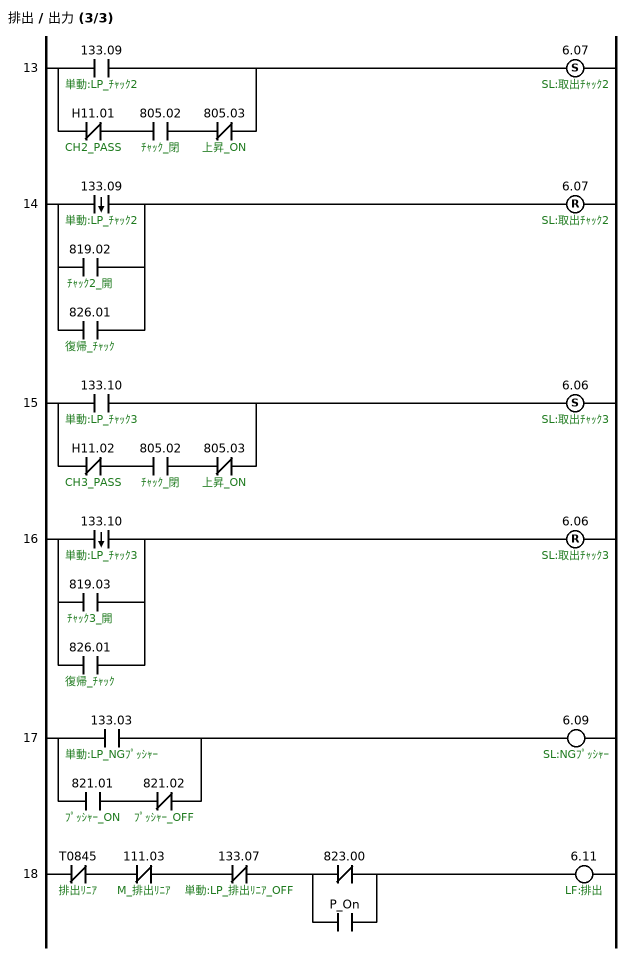
; [picture p192: 排出 / 出力, rungs 13-18]
; rung 13
LD 133.09  ; 単動:LP_ﾁｬｯｸ2
LDNOT H11.01  ; CH2_PASS
AND 805.02  ; ﾁｬｯｸ_閉
ANDNOT 805.03  ; 上昇_ON
ORLD
SET 6.07  ; SL:取出ﾁｬｯｸ2
; rung 14
%LD 133.09  ; 単動:LP_ﾁｬｯｸ2
OR 819.02  ; ﾁｬｯｸ2_開
OR 826.01  ; 復帰_ﾁｬｯｸ
RSET 6.07  ; SL:取出ﾁｬｯｸ2
; rung 15
LD 133.10  ; 単動:LP_ﾁｬｯｸ3
LDNOT H11.02  ; CH3_PASS
AND 805.02  ; ﾁｬｯｸ_閉
ANDNOT 805.03  ; 上昇_ON
ORLD
SET 6.06  ; SL:取出ﾁｬｯｸ3
; rung 16
%LD 133.10  ; 単動:LP_ﾁｬｯｸ3
OR 819.03  ; ﾁｬｯｸ3_開
OR 826.01  ; 復帰_ﾁｬｯｸ
RSET 6.06  ; SL:取出ﾁｬｯｸ3
; rung 17
LD 133.03  ; 単動:LP_NGﾌﾟｯｼｬｰ
LD 821.01  ; ﾌﾟｯｼｬｰ_ON
ANDNOT 821.02  ; ﾌﾟｯｼｬｰ_OFF
ORLD
OUT 6.09  ; SL:NGﾌﾟｯｼｬｰ
; rung 18
LDNOT T0845  ; 排出ﾘﾆｱ
ANDNOT 111.03  ; M_排出ﾘﾆｱ
ANDNOT 133.07  ; 単動:LP_排出ﾘﾆｱ_OFF
LDNOT 823.00
OR P_On
ANDLD
OUT 6.11  ; LF:排出

### Section ｴﾗｰ

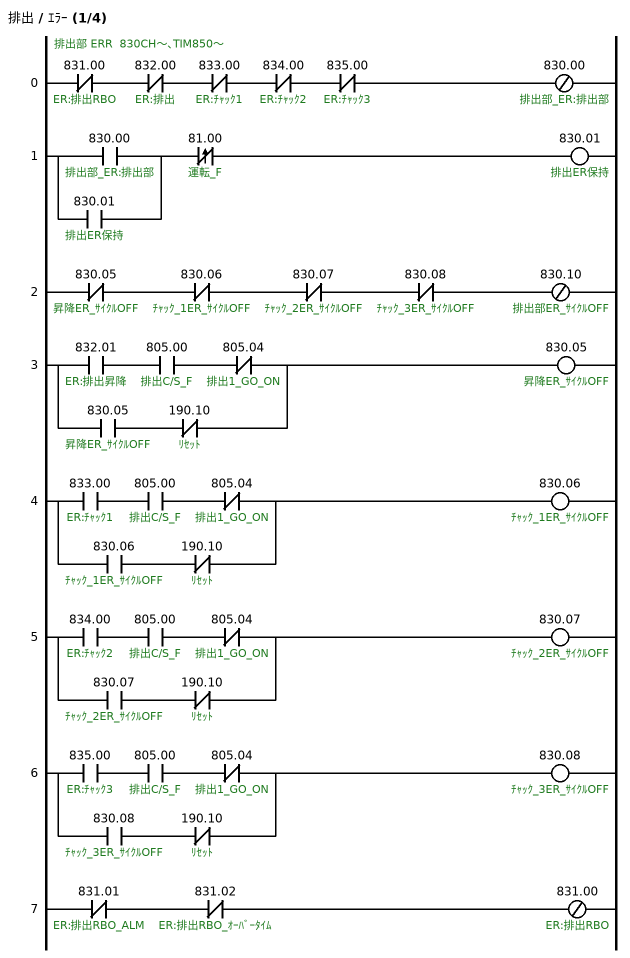
; rung 0: 排出部 ERR  830CH～､TIM850～
LDNOT 831.00  ; ER:排出RBO
ANDNOT 832.00  ; ER:排出
ANDNOT 833.00  ; ER:ﾁｬｯｸ1
ANDNOT 834.00  ; ER:ﾁｬｯｸ2
ANDNOT 835.00  ; ER:ﾁｬｯｸ3
OUTNOT 830.00  ; 排出部_ER:排出部
; rung 1
LD 830.00  ; 排出部_ER:排出部
OR 830.01  ; 排出ER保持
@ANDNOT 81.00  ; 運転_F
OUT 830.01  ; 排出ER保持
; rung 2
LDNOT 830.05  ; 昇降ER_ｻｲｸﾙOFF
ANDNOT 830.06  ; ﾁｬｯｸ_1ER_ｻｲｸﾙOFF
ANDNOT 830.07  ; ﾁｬｯｸ_2ER_ｻｲｸﾙOFF
ANDNOT 830.08  ; ﾁｬｯｸ_3ER_ｻｲｸﾙOFF
OUTNOT 830.10  ; 排出部ER_ｻｲｸﾙOFF
; rung 3
LD 832.01  ; ER:排出昇降
AND 805.00  ; 排出C/S_F
ANDNOT 805.04  ; 排出1_GO_ON
LD 830.05  ; 昇降ER_ｻｲｸﾙOFF
ANDNOT 190.10  ; ﾘｾｯﾄ
ORLD
OUT 830.05  ; 昇降ER_ｻｲｸﾙOFF
; rung 4
LD 833.00  ; ER:ﾁｬｯｸ1
AND 805.00  ; 排出C/S_F
ANDNOT 805.04  ; 排出1_GO_ON
LD 830.06  ; ﾁｬｯｸ_1ER_ｻｲｸﾙOFF
ANDNOT 190.10  ; ﾘｾｯﾄ
ORLD
OUT 830.06  ; ﾁｬｯｸ_1ER_ｻｲｸﾙOFF
; rung 5
LD 834.00  ; ER:ﾁｬｯｸ2
AND 805.00  ; 排出C/S_F
ANDNOT 805.04  ; 排出1_GO_ON
LD 830.07  ; ﾁｬｯｸ_2ER_ｻｲｸﾙOFF
ANDNOT 190.10  ; ﾘｾｯﾄ
ORLD
OUT 830.07  ; ﾁｬｯｸ_2ER_ｻｲｸﾙOFF
; rung 6
LD 835.00  ; ER:ﾁｬｯｸ3
AND 805.00  ; 排出C/S_F
ANDNOT 805.04  ; 排出1_GO_ON
LD 830.08  ; ﾁｬｯｸ_3ER_ｻｲｸﾙOFF
ANDNOT 190.10  ; ﾘｾｯﾄ
ORLD
OUT 830.08  ; ﾁｬｯｸ_3ER_ｻｲｸﾙOFF
; rung 7
LDNOT 831.01  ; ER:排出RBO_ALM
ANDNOT 831.02  ; ER:排出RBO_ｵｰﾊﾞｰﾀｲﾑ
OUTNOT 831.00  ; ER:排出RBO

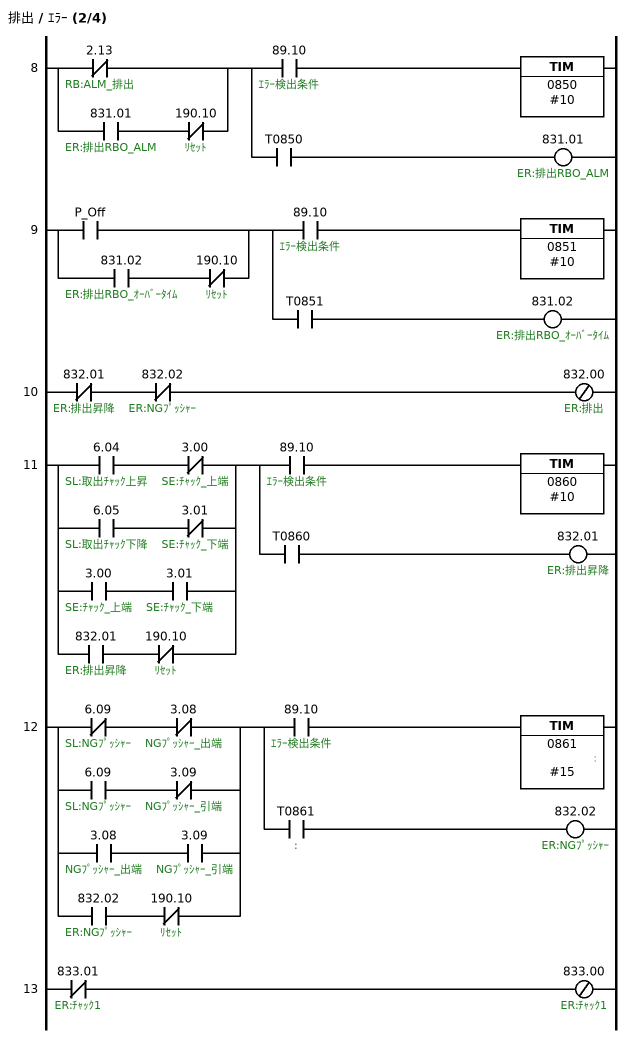
; rung 8
LDNOT 2.13  ; RB:ALM_排出
LD 831.01  ; ER:排出RBO_ALM
ANDNOT 190.10  ; ﾘｾｯﾄ
ORLD
OUT TR0
AND 89.10  ; ｴﾗｰ検出条件
TIM 0850 #10
LD TR0
AND T0850
OUT 831.01  ; ER:排出RBO_ALM
; rung 9
LD P_Off
LD 831.02  ; ER:排出RBO_ｵｰﾊﾞｰﾀｲﾑ
ANDNOT 190.10  ; ﾘｾｯﾄ
ORLD
OUT TR0
AND 89.10  ; ｴﾗｰ検出条件
TIM 0851 #10
LD TR0
AND T0851
OUT 831.02  ; ER:排出RBO_ｵｰﾊﾞｰﾀｲﾑ
; rung 10
LDNOT 832.01  ; ER:排出昇降
ANDNOT 832.02  ; ER:NGﾌﾟｯｼｬｰ
OUTNOT 832.00  ; ER:排出
; rung 11
LD 6.04  ; SL:取出ﾁｬｯｸ上昇
ANDNOT 3.00  ; SE:ﾁｬｯｸ_上端
LD 6.05  ; SL:取出ﾁｬｯｸ下降
ANDNOT 3.01  ; SE:ﾁｬｯｸ_下端
ORLD
LD 3.00  ; SE:ﾁｬｯｸ_上端
AND 3.01  ; SE:ﾁｬｯｸ_下端
ORLD
LD 832.01  ; ER:排出昇降
ANDNOT 190.10  ; ﾘｾｯﾄ
ORLD
OUT TR0
AND 89.10  ; ｴﾗｰ検出条件
TIM 0860 #10
LD TR0
AND T0860
OUT 832.01  ; ER:排出昇降
; rung 12
LDNOT 6.09  ; SL:NGﾌﾟｯｼｬｰ
ANDNOT 3.08  ; NGﾌﾟｯｼｬｰ_出端
LD 6.09  ; SL:NGﾌﾟｯｼｬｰ
ANDNOT 3.09  ; NGﾌﾟｯｼｬｰ_引端
ORLD
LD 3.08  ; NGﾌﾟｯｼｬｰ_出端
AND 3.09  ; NGﾌﾟｯｼｬｰ_引端
ORLD
LD 832.02  ; ER:NGﾌﾟｯｼｬｰ
ANDNOT 190.10  ; ﾘｾｯﾄ
ORLD
OUT TR0
AND 89.10  ; ｴﾗｰ検出条件
TIM 0861 #15  ; :
LD TR0
AND T0861  ; :
OUT 832.02  ; ER:NGﾌﾟｯｼｬｰ
; rung 13
LDNOT 833.01  ; ER:ﾁｬｯｸ1
OUTNOT 833.00  ; ER:ﾁｬｯｸ1

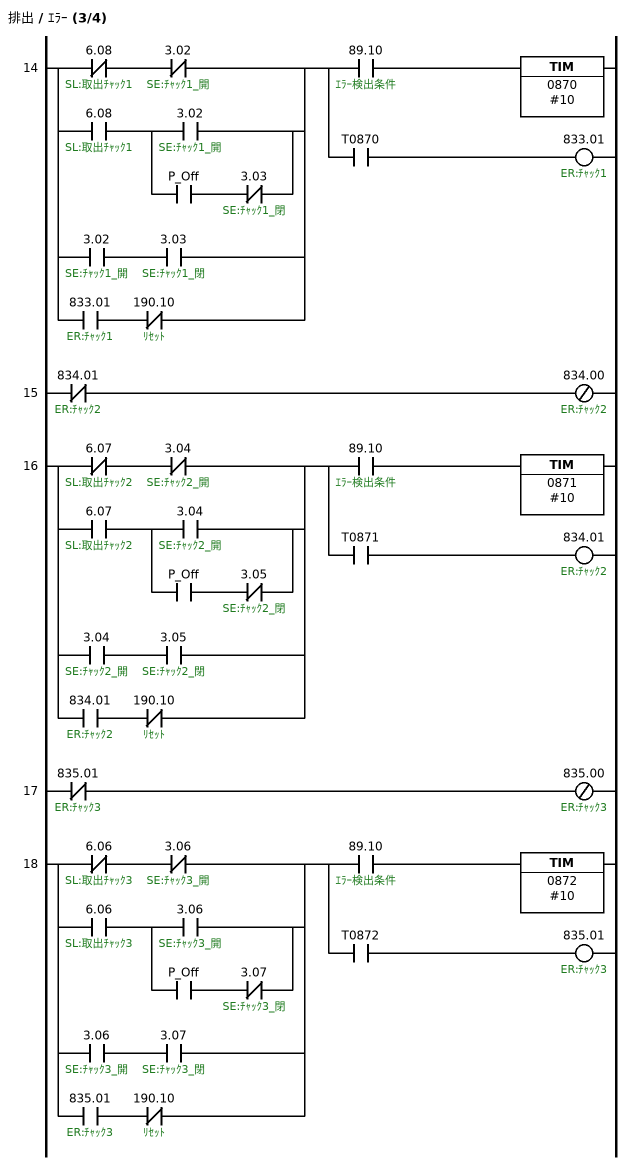
; rung 14
LDNOT 6.08  ; SL:取出ﾁｬｯｸ1
ANDNOT 3.02  ; SE:ﾁｬｯｸ1_開
LD 6.08  ; SL:取出ﾁｬｯｸ1
LD 3.02  ; SE:ﾁｬｯｸ1_開
LD P_Off
ANDNOT 3.03  ; SE:ﾁｬｯｸ1_閉
ORLD
ANDLD
ORLD
LD 3.02  ; SE:ﾁｬｯｸ1_開
AND 3.03  ; SE:ﾁｬｯｸ1_閉
ORLD
LD 833.01  ; ER:ﾁｬｯｸ1
ANDNOT 190.10  ; ﾘｾｯﾄ
ORLD
OUT TR0
AND 89.10  ; ｴﾗｰ検出条件
TIM 0870 #10
LD TR0
AND T0870
OUT 833.01  ; ER:ﾁｬｯｸ1
; rung 15
LDNOT 834.01  ; ER:ﾁｬｯｸ2
OUTNOT 834.00  ; ER:ﾁｬｯｸ2
; rung 16
LDNOT 6.07  ; SL:取出ﾁｬｯｸ2
ANDNOT 3.04  ; SE:ﾁｬｯｸ2_開
LD 6.07  ; SL:取出ﾁｬｯｸ2
LD 3.04  ; SE:ﾁｬｯｸ2_開
LD P_Off
ANDNOT 3.05  ; SE:ﾁｬｯｸ2_閉
ORLD
ANDLD
ORLD
LD 3.04  ; SE:ﾁｬｯｸ2_開
AND 3.05  ; SE:ﾁｬｯｸ2_閉
ORLD
LD 834.01  ; ER:ﾁｬｯｸ2
ANDNOT 190.10  ; ﾘｾｯﾄ
ORLD
OUT TR0
AND 89.10  ; ｴﾗｰ検出条件
TIM 0871 #10
LD TR0
AND T0871
OUT 834.01  ; ER:ﾁｬｯｸ2
; rung 17
LDNOT 835.01  ; ER:ﾁｬｯｸ3
OUTNOT 835.00  ; ER:ﾁｬｯｸ3
; rung 18
LDNOT 6.06  ; SL:取出ﾁｬｯｸ3
ANDNOT 3.06  ; SE:ﾁｬｯｸ3_開
LD 6.06  ; SL:取出ﾁｬｯｸ3
LD 3.06  ; SE:ﾁｬｯｸ3_開
LD P_Off
ANDNOT 3.07  ; SE:ﾁｬｯｸ3_閉
ORLD
ANDLD
ORLD
LD 3.06  ; SE:ﾁｬｯｸ3_開
AND 3.07  ; SE:ﾁｬｯｸ3_閉
ORLD
LD 835.01  ; ER:ﾁｬｯｸ3
ANDNOT 190.10  ; ﾘｾｯﾄ
ORLD
OUT TR0
AND 89.10  ; ｴﾗｰ検出条件
TIM 0872 #10
LD TR0
AND T0872
OUT 835.01  ; ER:ﾁｬｯｸ3

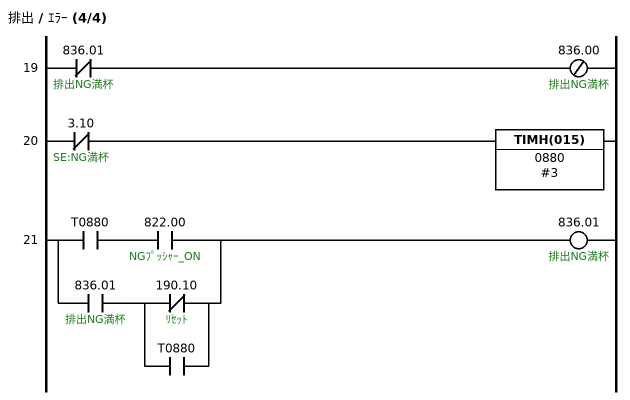
; rung 19
LDNOT 836.01  ; 排出NG満杯
OUTNOT 836.00  ; 排出NG満杯
; rung 20
LDNOT 3.10  ; SE:NG満杯
TIMH(015) 0880 #3
; rung 21
LD T0880
AND 822.00  ; NGﾌﾟｯｼｬｰ_ON
LD 836.01  ; 排出NG満杯
LDNOT 190.10  ; ﾘｾｯﾄ
OR T0880
ANDLD
ORLD
OUT 836.01  ; 排出NG満杯

### Section END
; rung 0
END(001)

## Program ﾃﾞｰﾀ収集 (cyclic task 8)

### Section 通信ST

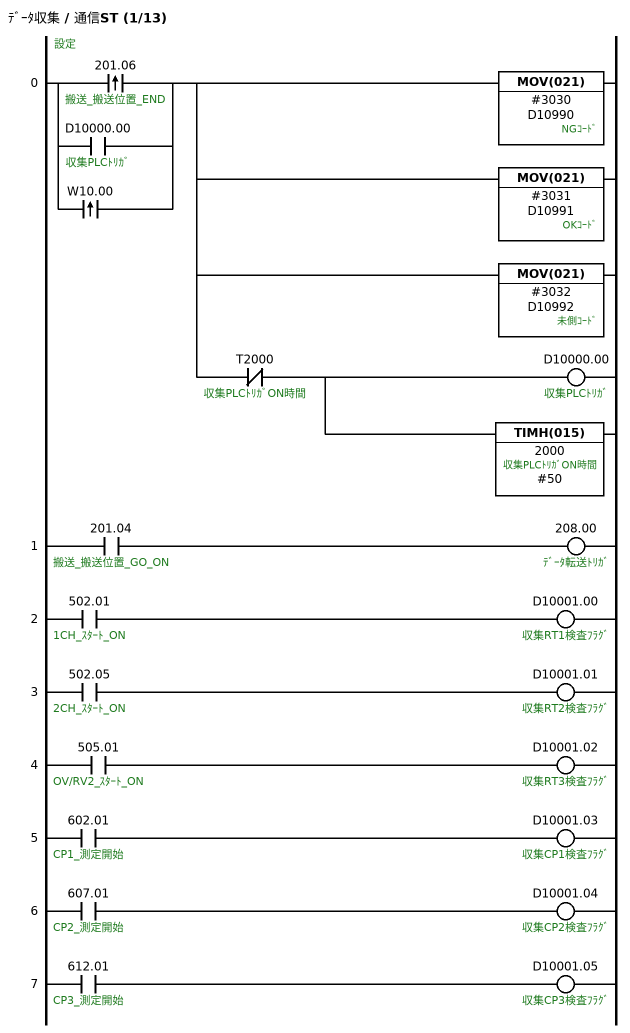
; rung 0: 設定
@LD 201.06  ; 搬送_搬送位置_END
OR D10000.00  ; 収集PLCﾄﾘｶﾞ
@OR W10.00
MOV(021) #3030 D10990  ; NGｺｰﾄﾞ
MOV(021) #3031 D10991  ; OKｺｰﾄﾞ
MOV(021) #3032 D10992  ; 未側ｺｰﾄﾞ
ANDNOT T2000  ; 収集PLCﾄﾘｶﾞON時間
OUT D10000.00  ; 収集PLCﾄﾘｶﾞ
TIMH(015) 2000 #50  ; 収集PLCﾄﾘｶﾞON時間
; rung 1
LD 201.04  ; 搬送_搬送位置_GO_ON
OUT 208.00  ; ﾃﾞｰﾀ転送ﾄﾘｶﾞ
; rung 2
LD 502.01  ; 1CH_ｽﾀｰﾄ_ON
OUT D10001.00  ; 収集RT1検査ﾌﾗｸﾞ
; rung 3
LD 502.05  ; 2CH_ｽﾀｰﾄ_ON
OUT D10001.01  ; 収集RT2検査ﾌﾗｸﾞ
; rung 4
LD 505.01  ; OV/RV2_ｽﾀｰﾄ_ON
OUT D10001.02  ; 収集RT3検査ﾌﾗｸﾞ
; rung 5
LD 602.01  ; CP1_測定開始
OUT D10001.03  ; 収集CP1検査ﾌﾗｸﾞ
; rung 6
LD 607.01  ; CP2_測定開始
OUT D10001.04  ; 収集CP2検査ﾌﾗｸﾞ
; rung 7
LD 612.01  ; CP3_測定開始
OUT D10001.05  ; 収集CP3検査ﾌﾗｸﾞ

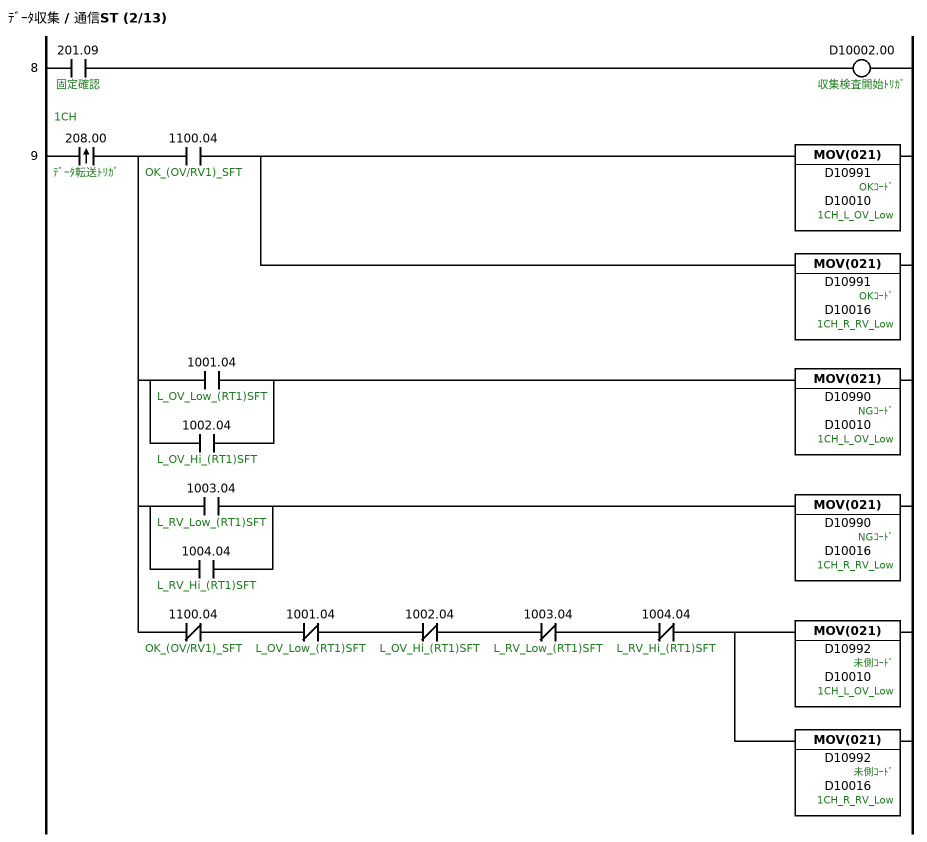
; rung 8
LD 201.09  ; 固定確認
OUT D10002.00  ; 収集検査開始ﾄﾘｶﾞ
; rung 9: 1CH
@LD 208.00  ; ﾃﾞｰﾀ転送ﾄﾘｶﾞ
OUT TR0
AND 1100.04  ; OK_(OV/RV1)_SFT
MOV(021) D10991 D10010  ; OKｺｰﾄﾞ, 1CH_L_OV_Low
MOV(021) D10991 D10016  ; OKｺｰﾄﾞ, 1CH_R_RV_Low
LD TR0
LD 1001.04  ; L_OV_Low_(RT1)SFT
OR 1002.04  ; L_OV_Hi_(RT1)SFT
ANDLD
MOV(021) D10990 D10010  ; NGｺｰﾄﾞ, 1CH_L_OV_Low
LD TR0
LD 1003.04  ; L_RV_Low_(RT1)SFT
OR 1004.04  ; L_RV_Hi_(RT1)SFT
ANDLD
MOV(021) D10990 D10016  ; NGｺｰﾄﾞ, 1CH_R_RV_Low
LD TR0
ANDNOT 1100.04  ; OK_(OV/RV1)_SFT
ANDNOT 1001.04  ; L_OV_Low_(RT1)SFT
ANDNOT 1002.04  ; L_OV_Hi_(RT1)SFT
ANDNOT 1003.04  ; L_RV_Low_(RT1)SFT
ANDNOT 1004.04  ; L_RV_Hi_(RT1)SFT
MOV(021) D10992 D10010  ; 未側ｺｰﾄﾞ, 1CH_L_OV_Low
MOV(021) D10992 D10016  ; 未側ｺｰﾄﾞ, 1CH_R_RV_Low

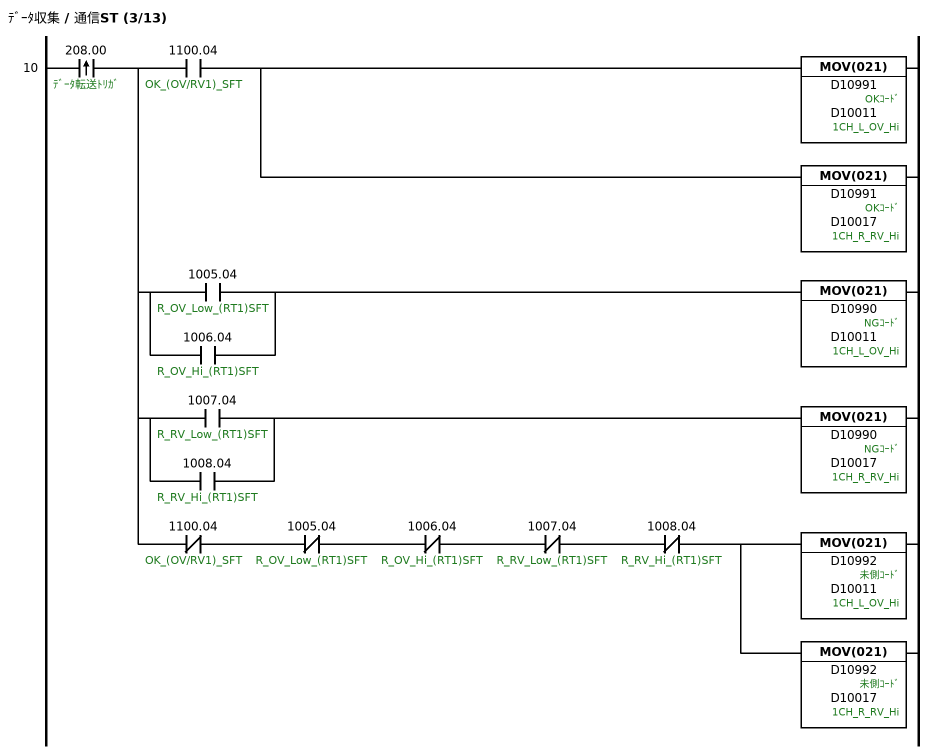
; rung 10
@LD 208.00  ; ﾃﾞｰﾀ転送ﾄﾘｶﾞ
OUT TR0
AND 1100.04  ; OK_(OV/RV1)_SFT
MOV(021) D10991 D10011  ; OKｺｰﾄﾞ, 1CH_L_OV_Hi
MOV(021) D10991 D10017  ; OKｺｰﾄﾞ, 1CH_R_RV_Hi
LD TR0
LD 1005.04  ; R_OV_Low_(RT1)SFT
OR 1006.04  ; R_OV_Hi_(RT1)SFT
ANDLD
MOV(021) D10990 D10011  ; NGｺｰﾄﾞ, 1CH_L_OV_Hi
LD TR0
LD 1007.04  ; R_RV_Low_(RT1)SFT
OR 1008.04  ; R_RV_Hi_(RT1)SFT
ANDLD
MOV(021) D10990 D10017  ; NGｺｰﾄﾞ, 1CH_R_RV_Hi
LD TR0
ANDNOT 1100.04  ; OK_(OV/RV1)_SFT
ANDNOT 1005.04  ; R_OV_Low_(RT1)SFT
ANDNOT 1006.04  ; R_OV_Hi_(RT1)SFT
ANDNOT 1007.04  ; R_RV_Low_(RT1)SFT
ANDNOT 1008.04  ; R_RV_Hi_(RT1)SFT
MOV(021) D10992 D10011  ; 未側ｺｰﾄﾞ, 1CH_L_OV_Hi
MOV(021) D10992 D10017  ; 未側ｺｰﾄﾞ, 1CH_R_RV_Hi

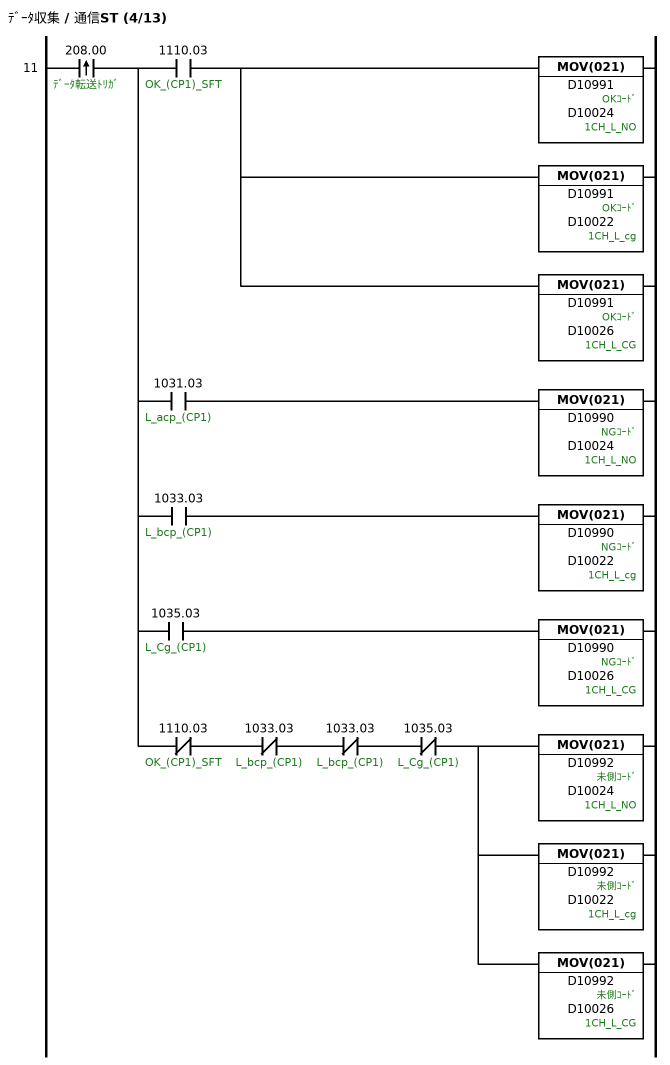
; rung 11
@LD 208.00  ; ﾃﾞｰﾀ転送ﾄﾘｶﾞ
OUT TR0
AND 1110.03  ; OK_(CP1)_SFT
MOV(021) D10991 D10024  ; OKｺｰﾄﾞ, 1CH_L_NO
MOV(021) D10991 D10022  ; OKｺｰﾄﾞ, 1CH_L_cg
MOV(021) D10991 D10026  ; OKｺｰﾄﾞ, 1CH_L_CG
LD TR0
AND 1031.03  ; L_acp_(CP1)
MOV(021) D10990 D10024  ; NGｺｰﾄﾞ, 1CH_L_NO
LD TR0
AND 1033.03  ; L_bcp_(CP1)
MOV(021) D10990 D10022  ; NGｺｰﾄﾞ, 1CH_L_cg
LD TR0
AND 1035.03  ; L_Cg_(CP1)
MOV(021) D10990 D10026  ; NGｺｰﾄﾞ, 1CH_L_CG
LD TR0
ANDNOT 1110.03  ; OK_(CP1)_SFT
ANDNOT 1033.03  ; L_bcp_(CP1)
ANDNOT 1033.03  ; L_bcp_(CP1)
ANDNOT 1035.03  ; L_Cg_(CP1)
MOV(021) D10992 D10024  ; 未側ｺｰﾄﾞ, 1CH_L_NO
MOV(021) D10992 D10022  ; 未側ｺｰﾄﾞ, 1CH_L_cg
MOV(021) D10992 D10026  ; 未側ｺｰﾄﾞ, 1CH_L_CG

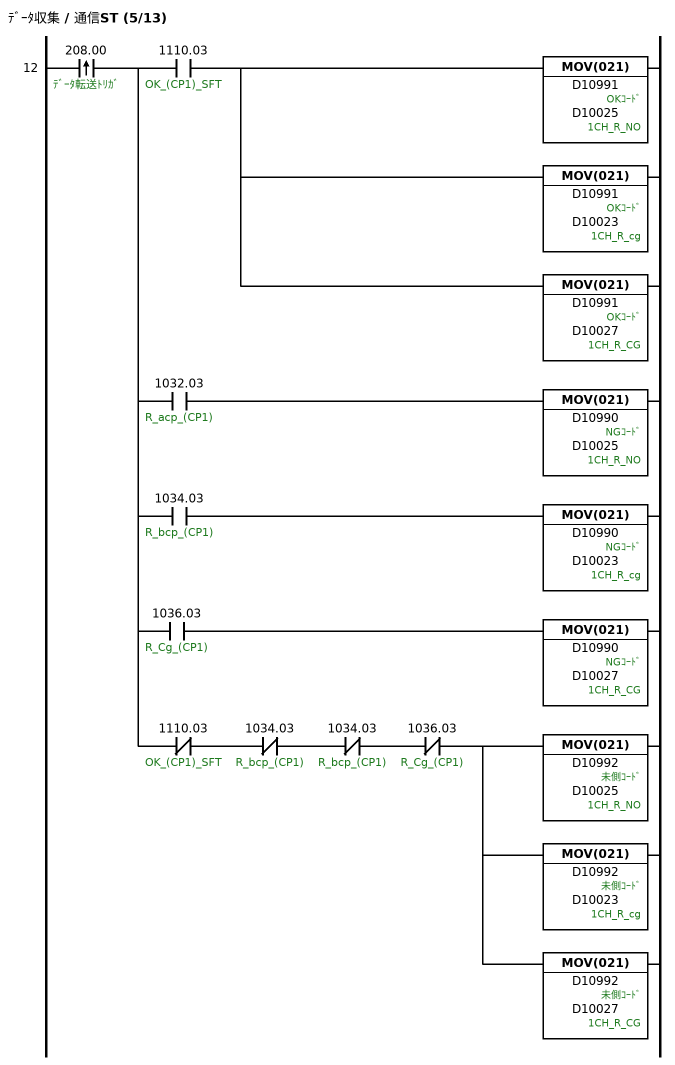
; rung 12
@LD 208.00  ; ﾃﾞｰﾀ転送ﾄﾘｶﾞ
OUT TR0
AND 1110.03  ; OK_(CP1)_SFT
MOV(021) D10991 D10025  ; OKｺｰﾄﾞ, 1CH_R_NO
MOV(021) D10991 D10023  ; OKｺｰﾄﾞ, 1CH_R_cg
MOV(021) D10991 D10027  ; OKｺｰﾄﾞ, 1CH_R_CG
LD TR0
AND 1032.03  ; R_acp_(CP1)
MOV(021) D10990 D10025  ; NGｺｰﾄﾞ, 1CH_R_NO
LD TR0
AND 1034.03  ; R_bcp_(CP1)
MOV(021) D10990 D10023  ; NGｺｰﾄﾞ, 1CH_R_cg
LD TR0
AND 1036.03  ; R_Cg_(CP1)
MOV(021) D10990 D10027  ; NGｺｰﾄﾞ, 1CH_R_CG
LD TR0
ANDNOT 1110.03  ; OK_(CP1)_SFT
ANDNOT 1034.03  ; R_bcp_(CP1)
ANDNOT 1034.03  ; R_bcp_(CP1)
ANDNOT 1036.03  ; R_Cg_(CP1)
MOV(021) D10992 D10025  ; 未側ｺｰﾄﾞ, 1CH_R_NO
MOV(021) D10992 D10023  ; 未側ｺｰﾄﾞ, 1CH_R_cg
MOV(021) D10992 D10027  ; 未側ｺｰﾄﾞ, 1CH_R_CG

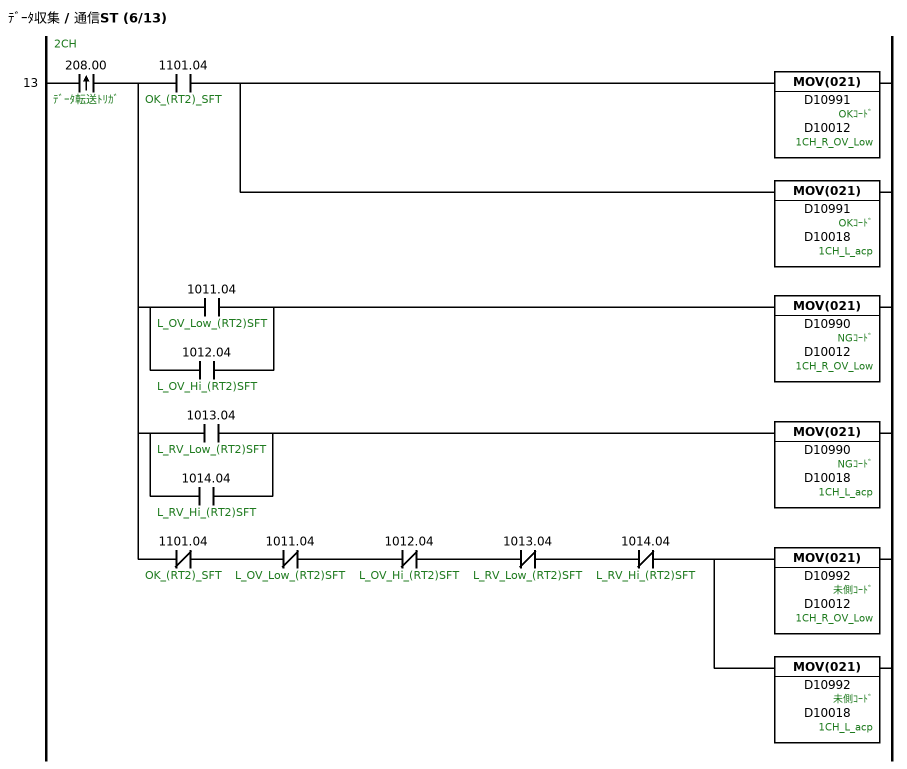
; rung 13: 2CH
@LD 208.00  ; ﾃﾞｰﾀ転送ﾄﾘｶﾞ
OUT TR0
AND 1101.04  ; OK_(RT2)_SFT
MOV(021) D10991 D10012  ; OKｺｰﾄﾞ, 1CH_R_OV_Low
MOV(021) D10991 D10018  ; OKｺｰﾄﾞ, 1CH_L_acp
LD TR0
LD 1011.04  ; L_OV_Low_(RT2)SFT
OR 1012.04  ; L_OV_Hi_(RT2)SFT
ANDLD
MOV(021) D10990 D10012  ; NGｺｰﾄﾞ, 1CH_R_OV_Low
LD TR0
LD 1013.04  ; L_RV_Low_(RT2)SFT
OR 1014.04  ; L_RV_Hi_(RT2)SFT
ANDLD
MOV(021) D10990 D10018  ; NGｺｰﾄﾞ, 1CH_L_acp
LD TR0
ANDNOT 1101.04  ; OK_(RT2)_SFT
ANDNOT 1011.04  ; L_OV_Low_(RT2)SFT
ANDNOT 1012.04  ; L_OV_Hi_(RT2)SFT
ANDNOT 1013.04  ; L_RV_Low_(RT2)SFT
ANDNOT 1014.04  ; L_RV_Hi_(RT2)SFT
MOV(021) D10992 D10012  ; 未側ｺｰﾄﾞ, 1CH_R_OV_Low
MOV(021) D10992 D10018  ; 未側ｺｰﾄﾞ, 1CH_L_acp

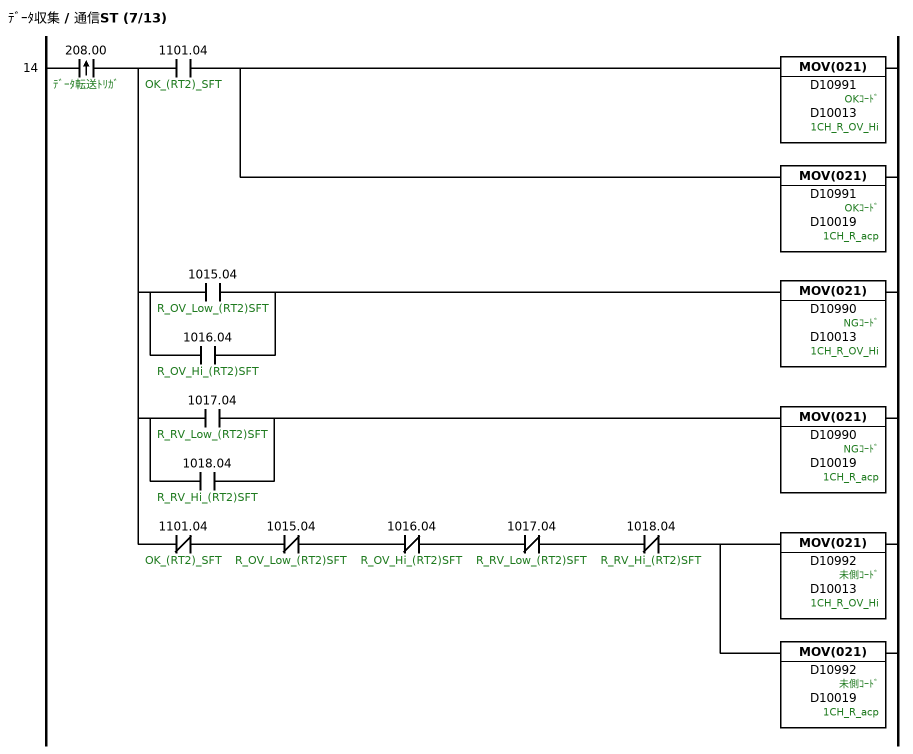
; rung 14
@LD 208.00  ; ﾃﾞｰﾀ転送ﾄﾘｶﾞ
OUT TR0
AND 1101.04  ; OK_(RT2)_SFT
MOV(021) D10991 D10013  ; OKｺｰﾄﾞ, 1CH_R_OV_Hi
MOV(021) D10991 D10019  ; OKｺｰﾄﾞ, 1CH_R_acp
LD TR0
LD 1015.04  ; R_OV_Low_(RT2)SFT
OR 1016.04  ; R_OV_Hi_(RT2)SFT
ANDLD
MOV(021) D10990 D10013  ; NGｺｰﾄﾞ, 1CH_R_OV_Hi
LD TR0
LD 1017.04  ; R_RV_Low_(RT2)SFT
OR 1018.04  ; R_RV_Hi_(RT2)SFT
ANDLD
MOV(021) D10990 D10019  ; NGｺｰﾄﾞ, 1CH_R_acp
LD TR0
ANDNOT 1101.04  ; OK_(RT2)_SFT
ANDNOT 1015.04  ; R_OV_Low_(RT2)SFT
ANDNOT 1016.04  ; R_OV_Hi_(RT2)SFT
ANDNOT 1017.04  ; R_RV_Low_(RT2)SFT
ANDNOT 1018.04  ; R_RV_Hi_(RT2)SFT
MOV(021) D10992 D10013  ; 未側ｺｰﾄﾞ, 1CH_R_OV_Hi
MOV(021) D10992 D10019  ; 未側ｺｰﾄﾞ, 1CH_R_acp

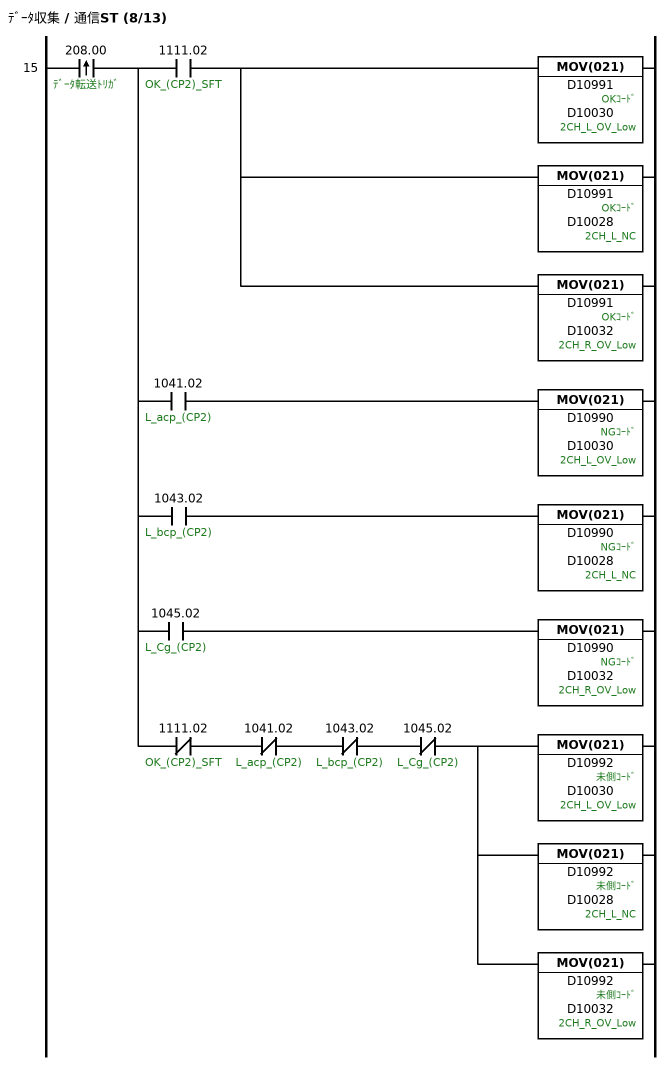
; rung 15
@LD 208.00  ; ﾃﾞｰﾀ転送ﾄﾘｶﾞ
OUT TR0
AND 1111.02  ; OK_(CP2)_SFT
MOV(021) D10991 D10030  ; OKｺｰﾄﾞ, 2CH_L_OV_Low
MOV(021) D10991 D10028  ; OKｺｰﾄﾞ, 2CH_L_NC
MOV(021) D10991 D10032  ; OKｺｰﾄﾞ, 2CH_R_OV_Low
LD TR0
AND 1041.02  ; L_acp_(CP2)
MOV(021) D10990 D10030  ; NGｺｰﾄﾞ, 2CH_L_OV_Low
LD TR0
AND 1043.02  ; L_bcp_(CP2)
MOV(021) D10990 D10028  ; NGｺｰﾄﾞ, 2CH_L_NC
LD TR0
AND 1045.02  ; L_Cg_(CP2)
MOV(021) D10990 D10032  ; NGｺｰﾄﾞ, 2CH_R_OV_Low
LD TR0
ANDNOT 1111.02  ; OK_(CP2)_SFT
ANDNOT 1041.02  ; L_acp_(CP2)
ANDNOT 1043.02  ; L_bcp_(CP2)
ANDNOT 1045.02  ; L_Cg_(CP2)
MOV(021) D10992 D10030  ; 未側ｺｰﾄﾞ, 2CH_L_OV_Low
MOV(021) D10992 D10028  ; 未側ｺｰﾄﾞ, 2CH_L_NC
MOV(021) D10992 D10032  ; 未側ｺｰﾄﾞ, 2CH_R_OV_Low

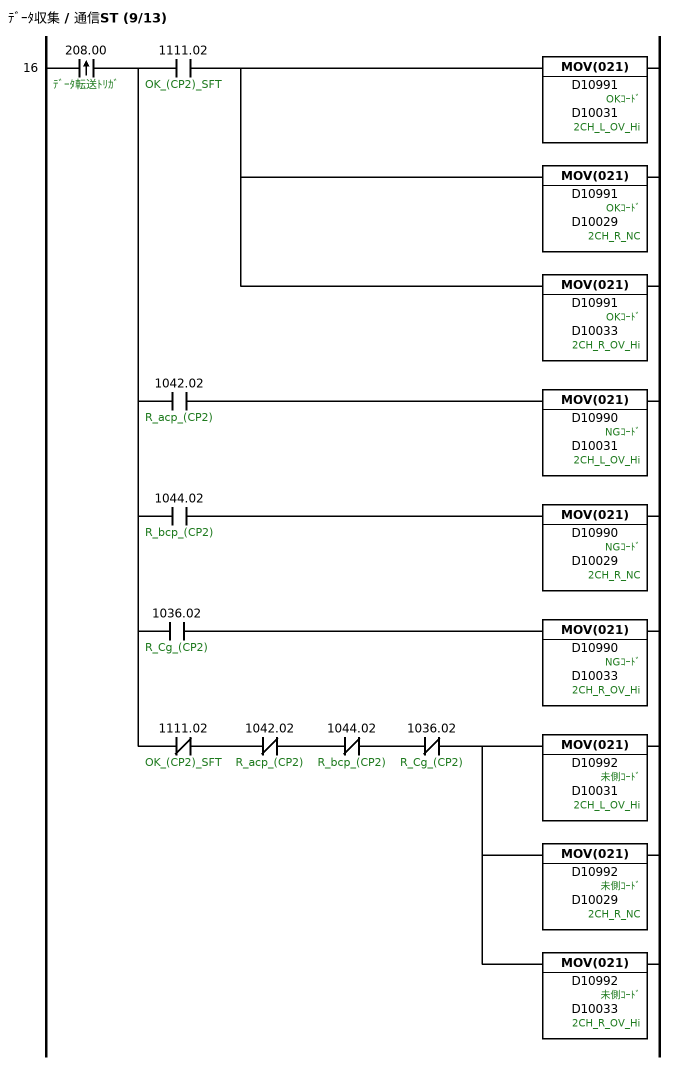
; rung 16
@LD 208.00  ; ﾃﾞｰﾀ転送ﾄﾘｶﾞ
OUT TR0
AND 1111.02  ; OK_(CP2)_SFT
MOV(021) D10991 D10031  ; OKｺｰﾄﾞ, 2CH_L_OV_Hi
MOV(021) D10991 D10029  ; OKｺｰﾄﾞ, 2CH_R_NC
MOV(021) D10991 D10033  ; OKｺｰﾄﾞ, 2CH_R_OV_Hi
LD TR0
AND 1042.02  ; R_acp_(CP2)
MOV(021) D10990 D10031  ; NGｺｰﾄﾞ, 2CH_L_OV_Hi
LD TR0
AND 1044.02  ; R_bcp_(CP2)
MOV(021) D10990 D10029  ; NGｺｰﾄﾞ, 2CH_R_NC
LD TR0
AND 1036.02  ; R_Cg_(CP2)
MOV(021) D10990 D10033  ; NGｺｰﾄﾞ, 2CH_R_OV_Hi
LD TR0
ANDNOT 1111.02  ; OK_(CP2)_SFT
ANDNOT 1042.02  ; R_acp_(CP2)
ANDNOT 1044.02  ; R_bcp_(CP2)
ANDNOT 1036.02  ; R_Cg_(CP2)
MOV(021) D10992 D10031  ; 未側ｺｰﾄﾞ, 2CH_L_OV_Hi
MOV(021) D10992 D10029  ; 未側ｺｰﾄﾞ, 2CH_R_NC
MOV(021) D10992 D10033  ; 未側ｺｰﾄﾞ, 2CH_R_OV_Hi

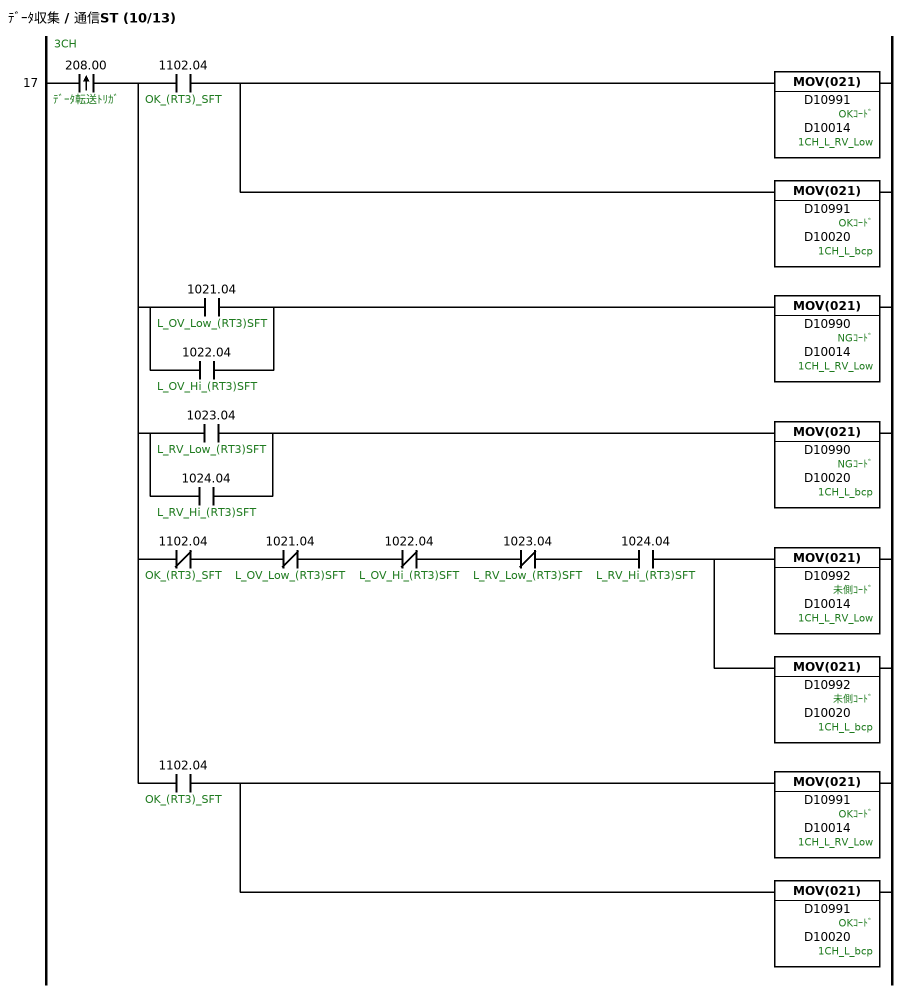
; rung 17: 3CH
@LD 208.00  ; ﾃﾞｰﾀ転送ﾄﾘｶﾞ
OUT TR0
AND 1102.04  ; OK_(RT3)_SFT
MOV(021) D10991 D10014  ; OKｺｰﾄﾞ, 1CH_L_RV_Low
MOV(021) D10991 D10020  ; OKｺｰﾄﾞ, 1CH_L_bcp
LD TR0
LD 1021.04  ; L_OV_Low_(RT3)SFT
OR 1022.04  ; L_OV_Hi_(RT3)SFT
ANDLD
MOV(021) D10990 D10014  ; NGｺｰﾄﾞ, 1CH_L_RV_Low
LD TR0
LD 1023.04  ; L_RV_Low_(RT3)SFT
OR 1024.04  ; L_RV_Hi_(RT3)SFT
ANDLD
MOV(021) D10990 D10020  ; NGｺｰﾄﾞ, 1CH_L_bcp
LD TR0
ANDNOT 1102.04  ; OK_(RT3)_SFT
ANDNOT 1021.04  ; L_OV_Low_(RT3)SFT
ANDNOT 1022.04  ; L_OV_Hi_(RT3)SFT
ANDNOT 1023.04  ; L_RV_Low_(RT3)SFT
AND 1024.04  ; L_RV_Hi_(RT3)SFT
MOV(021) D10992 D10014  ; 未側ｺｰﾄﾞ, 1CH_L_RV_Low
MOV(021) D10992 D10020  ; 未側ｺｰﾄﾞ, 1CH_L_bcp
LD TR0
AND 1102.04  ; OK_(RT3)_SFT
MOV(021) D10991 D10014  ; OKｺｰﾄﾞ, 1CH_L_RV_Low
MOV(021) D10991 D10020  ; OKｺｰﾄﾞ, 1CH_L_bcp

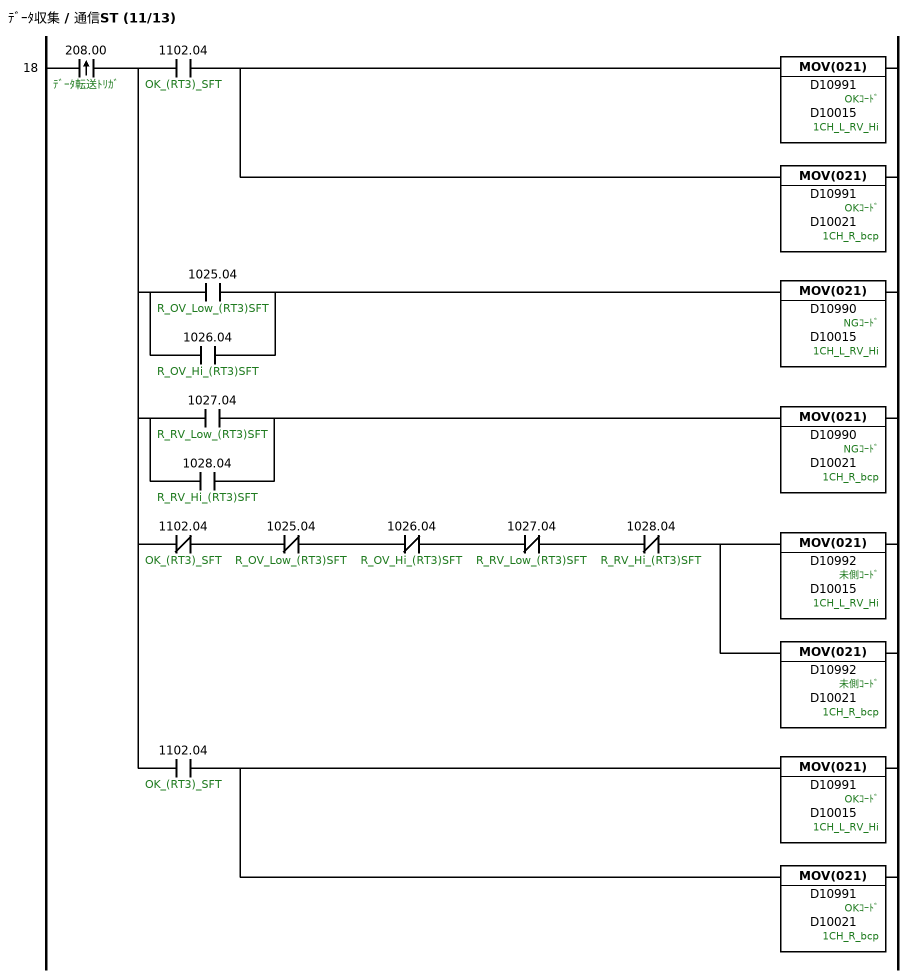
; rung 18
@LD 208.00  ; ﾃﾞｰﾀ転送ﾄﾘｶﾞ
OUT TR0
AND 1102.04  ; OK_(RT3)_SFT
MOV(021) D10991 D10015  ; OKｺｰﾄﾞ, 1CH_L_RV_Hi
MOV(021) D10991 D10021  ; OKｺｰﾄﾞ, 1CH_R_bcp
LD TR0
LD 1025.04  ; R_OV_Low_(RT3)SFT
OR 1026.04  ; R_OV_Hi_(RT3)SFT
ANDLD
MOV(021) D10990 D10015  ; NGｺｰﾄﾞ, 1CH_L_RV_Hi
LD TR0
LD 1027.04  ; R_RV_Low_(RT3)SFT
OR 1028.04  ; R_RV_Hi_(RT3)SFT
ANDLD
MOV(021) D10990 D10021  ; NGｺｰﾄﾞ, 1CH_R_bcp
LD TR0
ANDNOT 1102.04  ; OK_(RT3)_SFT
ANDNOT 1025.04  ; R_OV_Low_(RT3)SFT
ANDNOT 1026.04  ; R_OV_Hi_(RT3)SFT
ANDNOT 1027.04  ; R_RV_Low_(RT3)SFT
ANDNOT 1028.04  ; R_RV_Hi_(RT3)SFT
MOV(021) D10992 D10015  ; 未側ｺｰﾄﾞ, 1CH_L_RV_Hi
MOV(021) D10992 D10021  ; 未側ｺｰﾄﾞ, 1CH_R_bcp
LD TR0
AND 1102.04  ; OK_(RT3)_SFT
MOV(021) D10991 D10015  ; OKｺｰﾄﾞ, 1CH_L_RV_Hi
MOV(021) D10991 D10021  ; OKｺｰﾄﾞ, 1CH_R_bcp

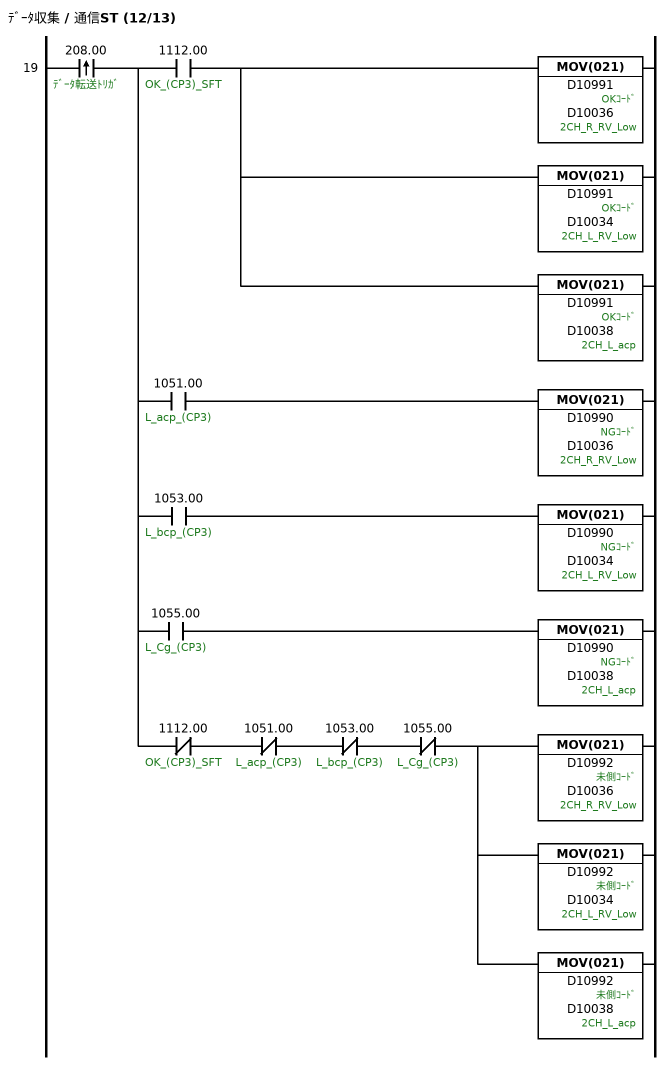
; rung 19
@LD 208.00  ; ﾃﾞｰﾀ転送ﾄﾘｶﾞ
OUT TR0
AND 1112.00  ; OK_(CP3)_SFT
MOV(021) D10991 D10036  ; OKｺｰﾄﾞ, 2CH_R_RV_Low
MOV(021) D10991 D10034  ; OKｺｰﾄﾞ, 2CH_L_RV_Low
MOV(021) D10991 D10038  ; OKｺｰﾄﾞ, 2CH_L_acp
LD TR0
AND 1051.00  ; L_acp_(CP3)
MOV(021) D10990 D10036  ; NGｺｰﾄﾞ, 2CH_R_RV_Low
LD TR0
AND 1053.00  ; L_bcp_(CP3)
MOV(021) D10990 D10034  ; NGｺｰﾄﾞ, 2CH_L_RV_Low
LD TR0
AND 1055.00  ; L_Cg_(CP3)
MOV(021) D10990 D10038  ; NGｺｰﾄﾞ, 2CH_L_acp
LD TR0
ANDNOT 1112.00  ; OK_(CP3)_SFT
ANDNOT 1051.00  ; L_acp_(CP3)
ANDNOT 1053.00  ; L_bcp_(CP3)
ANDNOT 1055.00  ; L_Cg_(CP3)
MOV(021) D10992 D10036  ; 未側ｺｰﾄﾞ, 2CH_R_RV_Low
MOV(021) D10992 D10034  ; 未側ｺｰﾄﾞ, 2CH_L_RV_Low
MOV(021) D10992 D10038  ; 未側ｺｰﾄﾞ, 2CH_L_acp

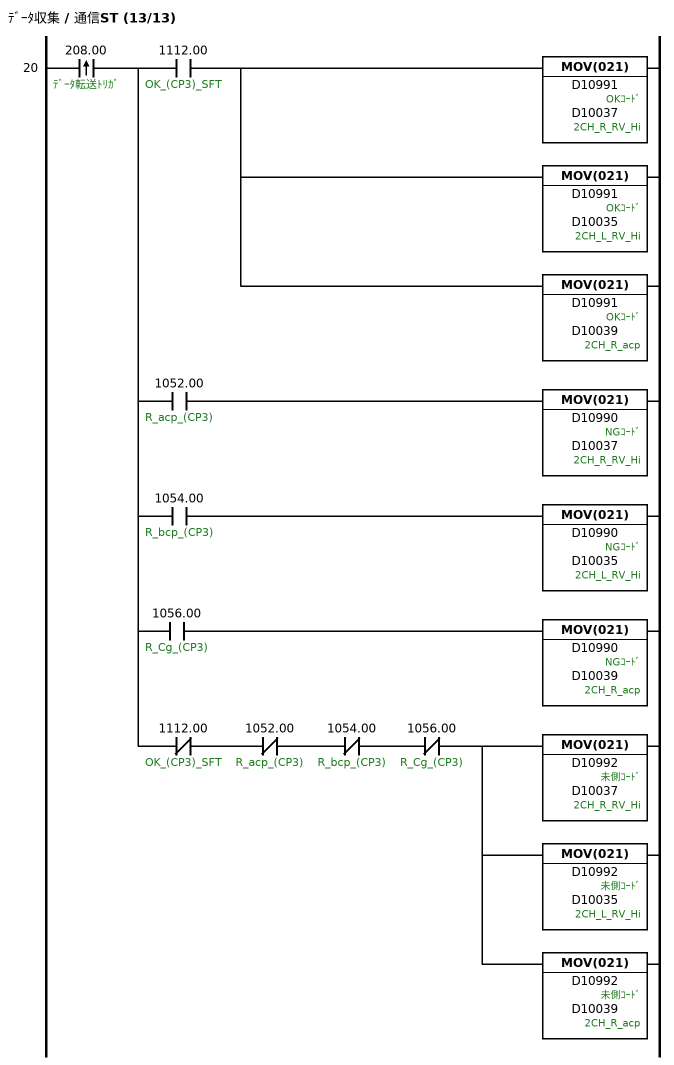
; rung 20
@LD 208.00  ; ﾃﾞｰﾀ転送ﾄﾘｶﾞ
OUT TR0
AND 1112.00  ; OK_(CP3)_SFT
MOV(021) D10991 D10037  ; OKｺｰﾄﾞ, 2CH_R_RV_Hi
MOV(021) D10991 D10035  ; OKｺｰﾄﾞ, 2CH_L_RV_Hi
MOV(021) D10991 D10039  ; OKｺｰﾄﾞ, 2CH_R_acp
LD TR0
AND 1052.00  ; R_acp_(CP3)
MOV(021) D10990 D10037  ; NGｺｰﾄﾞ, 2CH_R_RV_Hi
LD TR0
AND 1054.00  ; R_bcp_(CP3)
MOV(021) D10990 D10035  ; NGｺｰﾄﾞ, 2CH_L_RV_Hi
LD TR0
AND 1056.00  ; R_Cg_(CP3)
MOV(021) D10990 D10039  ; NGｺｰﾄﾞ, 2CH_R_acp
LD TR0
ANDNOT 1112.00  ; OK_(CP3)_SFT
ANDNOT 1052.00  ; R_acp_(CP3)
ANDNOT 1054.00  ; R_bcp_(CP3)
ANDNOT 1056.00  ; R_Cg_(CP3)
MOV(021) D10992 D10037  ; 未側ｺｰﾄﾞ, 2CH_R_RV_Hi
MOV(021) D10992 D10035  ; 未側ｺｰﾄﾞ, 2CH_L_RV_Hi
MOV(021) D10992 D10039  ; 未側ｺｰﾄﾞ, 2CH_R_acp

### Section END
; rung 0
END(001)